(* CODESYS project Opción de grado.project

Project tree, tasks and I/O mapping:
  Device : CODESYS Control Win V3 64, 3S - Smart Software Solutions GmbH, version 3.5.9.10
    application Application
      libraries: Standard, * (System)
      task MainTask (cyclic, interval t#20ms, priority 1) calls PLC_PRG
      var global PLC_PRG [ST]
*)

// Device/Application/PLC_PRG
VAR_GLOBAL

    (* CODESYS → FluidSIM In Module 1 *)
    Q_VENTOSA_OMEGA_ON   : BOOL; (* Bit 0 → 1M1 *)
    Q_VENTOSA_OMEGA_OFF  : BOOL; (* Bit 1 → 1M2 *)
    Q_VENTOSA_PALET_ON   : BOOL; (* Bit 2 → 2M1 *)
    Q_VENTOSA_PALET_OFF  : BOOL; (* Bit 3 → 2M2 *)

    (* FluidSIM Out Module 1 → CODESYS *)
    I_PRESION_OMEGA      : BOOL; (* Bit 0 - sensor vacío Omega *)
    I_PRESION_PALET      : BOOL; (* Bit 1 - sensor vacío Palet *)

    (* Control general *)
    START                : BOOL;
    STOP                 : BOOL;
    EMERGENCIA           : BOOL;

    (* Estados internos *)
    SISTEMA_ACTIVO       : BOOL;
    VENTOSA_OMEGA_ACTIVA : BOOL;
    VENTOSA_PALET_ACTIVA : BOOL;

END_VAR
